(* IEC 61131-3 sources: Lasal/CPU_5344_V01/Class/IFM2400Input, 1 file *)

(* ---- IFM2400Input.st ---- *)
(*!
<Class
	Name               = "IFM2400Input"
	Revision           = "0.0"
	RealtimeTask       = "false"
	CyclicTask         = "true"
	DefCyclictime      = "2 ms"
	BackgroundTask     = "false"
	Sigmatek           = "false"
	OSInterface        = "false"
	HighPriority       = "false"
	Automatic          = "false"
	UpdateMode         = "Prescan"
	SharedCommandTable = "true"
	Objectsize         = "(660,1200)">
	<Channels>
		<Server Name="ActualMode" Visualized="true" Remotely="true" Initialize="false" WriteProtected="true" Retentive="false" Comment="Shows the currently active mode of the device (is only valid when the ClassState is _ClassOk and the FaultFlags are on _NoFault)"/>
		<Server Name="ClassState" Class="SDCIDevice" Visualized="true" Remotely="true" Initialize="false" WriteProtected="true" Retentive="false" Comment="Shows the current Status of the Hardware Class"/>
		<Server Name="ClassSvr" Visualized="false" Initialize="false" WriteProtected="true" Retentive="false"/>
		<Server Name="Input1" Visualized="false" Initialize="false" WriteProtected="true" Retentive="false"/>
		<Server Name="Input10" Visualized="false" Initialize="false" WriteProtected="true" Retentive="false"/>
		<Server Name="Input11" Visualized="false" Initialize="false" WriteProtected="true" Retentive="false"/>
		<Server Name="Input12" Visualized="false" Initialize="false" WriteProtected="true" Retentive="false"/>
		<Server Name="Input13" Visualized="false" Initialize="false" WriteProtected="true" Retentive="false"/>
		<Server Name="Input14" Visualized="false" Initialize="false" WriteProtected="true" Retentive="false"/>
		<Server Name="Input15" Visualized="false" Initialize="false" WriteProtected="true" Retentive="false"/>
		<Server Name="Input16" Visualized="false" Initialize="false" WriteProtected="true" Retentive="false"/>
		<Server Name="Input2" Visualized="false" Initialize="false" WriteProtected="true" Retentive="false"/>
		<Server Name="Input3" Visualized="false" Initialize="false" WriteProtected="true" Retentive="false"/>
		<Server Name="Input4" Visualized="false" Initialize="false" WriteProtected="true" Retentive="false"/>
		<Server Name="Input5" Visualized="false" Initialize="false" WriteProtected="true" Retentive="false"/>
		<Server Name="Input6" Visualized="false" Initialize="false" WriteProtected="true" Retentive="false"/>
		<Server Name="Input7" Visualized="false" Initialize="false" WriteProtected="true" Retentive="false"/>
		<Server Name="Input8" Visualized="false" Initialize="false" WriteProtected="true" Retentive="false"/>
		<Server Name="Input9" Visualized="false" Initialize="false" WriteProtected="true" Retentive="false"/>
		<Client Name="SDCIClass" Required="true" Internal="true"/>
		<Client Name="SdciIn" Required="true" Internal="false"/>
	</Channels>
	<Network Name="IFM2400Input">
		<!-- List of Components in this network -->
		<Components>
			<Object
				Name       = "SDCIClass"
				Class      = "SDCIClassIFM_AL2401"
				Position   = "(150,120)"
				Visualized = "true"
				Remotely   = "true">
				<Channels>
					<Server Name="ActualMode"/>
					<Server Name="ClassState"/>
					<Server Name="DeviceID"/>
					<Server Name="DirectInput"/>
					<Server Name="FaultFlags"/>
					<Server Name="Input"/>
					<Server Name="MinCycleTime"/>
					<Server Name="NbrOfEventsAvailable"/>
					<Server Name="Output"/>
					<Server Name="PortStateBits"/>
					<Server Name="VendorID"/>
					<Client Name="ReadPdoSize" Value="0"/>
					<Client Name="Required" Value="0"/>
					<Client Name="SdciIn"/>
					<Client Name="SkipEndianSwap" Value="0"/>
					<Client Name="StartUpMode" Value="_SDCI"/>
					<Client Name="WritePdoSize" Value="0"/>
				</Channels>
				<AdditionalData>
					<Entry Name="DeviceType" Value="SDCIClassIFM_AL2401"/>
				</AdditionalData>
			</Object>
		</Components>
		<Comments>
		</Comments>
		<!-- List of Connections in this network -->
		<Connections>
			<Connection Source="this.SDCIClass" Destination="SDCIClass.ClassState"/>
			<Connection Source="SDCIClass.SdciIn" Destination="this.SdciIn" Vertices="(150,210),(38,210),"/>
			<Connection Source="this.ClassState" Destination="SDCIClass.ClassState" Vertices="(990,270),(818,210),"/>
			<Connection Source="this.ActualMode" Destination="SDCIClass.ActualMode" Vertices="(990,330),(818,450),"/>
		</Connections>
		<!-- Headerfiles -->
		<Options>
		</Options>
	</Network>
</Class>
*)
IFM2400Input : CLASS
  //Servers:
	ClassSvr 	: SvrChCmd_DINT;
	ClassState 	: SvrChCmd_t_e_VaranErrors;
	ActualMode 	: SvrCh_t_SDCIPortMode_PTofCls_SdiasSDCIMaster;
	Input1 	: SvrCh_DINT;
	Input2 	: SvrCh_DINT;
	Input3 	: SvrCh_DINT;
	Input4 	: SvrCh_DINT;
	Input5 	: SvrCh_DINT;
	Input6 	: SvrCh_DINT;
	Input7 	: SvrCh_DINT;
	Input8 	: SvrCh_DINT;
	Input9 	: SvrCh_DINT;
	Input10 	: SvrCh_DINT;
	Input11 	: SvrCh_DINT;
	Input12 	: SvrCh_DINT;
	Input13 	: SvrCh_DINT;
	Input14 	: SvrCh_DINT;
	Input15 	: SvrCh_DINT;
	Input16 	: SvrCh_DINT;
  //Clients:
	SdciIn 	: CltChCmd_DINT;
	SDCIClass 	: CltChCmd_SDCIClassIFM_AL2401;
  //Variables:
		bdInputs : BDINT
		[
		];

  //Functions:

	FUNCTION VIRTUAL GLOBAL CyWork
		VAR_INPUT
			EAX 	: UDINT;
		END_VAR
		VAR_OUTPUT
			state (EAX) 	: UDINT;
		END_VAR;

	FUNCTION VIRTUAL GLOBAL ClassState::Read
		VAR_OUTPUT
			output (EAX) 	: t_e_VaranErrors;
		END_VAR;

	FUNCTION VIRTUAL GLOBAL ActualMode::Read
		VAR_OUTPUT
			output (EAX) 	: SdiasSDCIMaster::t_SDCIPortMode;
		END_VAR;
  //Tables:
	FUNCTION @STD
		VAR_OUTPUT
			ret_code	: CONFSTATES;
		END_VAR;
	FUNCTION GLOBAL TAB @CT_;
END_CLASS;

#pragma using SDCIClassIFM_AL2401

FUNCTION VIRTUAL GLOBAL IFM2400Input::CyWork
	VAR_INPUT
		EAX 	: UDINT;
	END_VAR
	VAR_OUTPUT
		state (EAX) 	: UDINT;
	END_VAR

  //read from io link from ifm splitterbox
  bdInputs := SDCIClass.GetReadPdoDWord(ReadOffset:=0);
  // if connection is ok
  if SDCIClass.ClassState = _ClassOk then
    // send inputs to servers
    Input1 := bdInputs.25;   // X1.0 - I1
    Input2 := bdInputs.17;   // X1.0 - I2
    Input3 := bdInputs.26;   // X1.1 - I1
    Input4 := bdInputs.18;   // X1.1 - I2
    Input5 := bdInputs.27;   // X1.2 - I1
    Input6 := bdInputs.19;   // X1.2 - I2
    Input7 := bdInputs.28;   // X1.3 - I1
    Input8 := bdInputs.20;   // X1.3 - I2

    Input9 := bdInputs.29;   // X1.4 - I1
    Input10 := bdInputs.21; // X1.4 - I2
    Input11 := bdInputs.30; // X1.5 - I1
    Input12 := bdInputs.22; // X1.5 - I2
    Input13 := bdInputs.31; // X1.6 - I1
    Input14 := bdInputs.23; // X1.6 - I2
    Input15 := bdInputs.32; // X1.7 - I1
    Input16 := bdInputs.24; // X1.7 - I2
  else
    // if no hardware, no inputs
    Input1 := 0;
    Input2 := 0;
    Input3 := 0;
    Input4 := 0;
    Input5 := 0;
    Input6 := 0;
    Input7 := 0;
    Input8 := 0;
    Input9 := 0;
    Input10:= 0;
    Input11 := 0;
    Input12 := 0;
    Input13 := 0;
    Input14 := 0;
    Input15 := 0;
    Input16 := 0;
  end_if;

	state := READY;

END_FUNCTION

FUNCTION VIRTUAL GLOBAL IFM2400Input::ClassState::Read
	VAR_OUTPUT
		output (EAX) 	: t_e_VaranErrors;
	END_VAR

	ClassState := SDCIClass.ClassState.Read();
	output := ClassState;

END_FUNCTION

FUNCTION VIRTUAL GLOBAL IFM2400Input::ActualMode::Read
	VAR_OUTPUT
		output (EAX) 	: SdiasSDCIMaster::t_SDCIPortMode;
	END_VAR

	ActualMode := SDCIClass.ActualMode.Read();
	output := ActualMode;

END_FUNCTION
